(* IEC 61131-3 sources: POMIRTS_lab3/AS/Library/AsHttp, 3 files *)

(* ---- AsHttp.typ ---- *)
(********************************************************************
 * COPYRIGHT -- Bernecker + Rainer
 ********************************************************************
 * Library: AsHttp
 * File: AsHttp.typ
 * Author: B+R
 ********************************************************************
 * Data types of library AsHttp
 ********************************************************************)

TYPE
	httpResponseHeader_t : 	STRUCT  (*response header structure*)
		protocol : STRING[20]; (*HTTP/1.0 or HTTP/1.1*)
		status : STRING[280]; (*HTTP status line e.g. "200 OK" , "404 Not Found"*)
		contentType : STRING[100]; (*MIME type specifying message body, e.g. "text/html"*)
		contentLength : UDINT; (*length of message data, should be equal to responseDataLen, optional input*)
		connection : STRING[80]; (*valid tokens are "Close" or "Keep-Alive", default is "Close"*)
		keepAlive : STRING[80]; (*e.g. "timeout=5, max=100", optional*)
		userLine : ARRAY[0..7]OF httpHeaderLine_t; (*userspecific headerlines, optional*)
		rawHeader : httpRawHeader_t; (*interface to add / get formatted headers, optional*)
	END_STRUCT;
	httpRequestHeader_t : 	STRUCT  (*request header structure*)
		protocol : STRING[20]; (*protocol version e.g. "HTTP/1.0" or "HTTP/1.1", optional input*)
		host : STRING[280]; (*host name or ip address of the server and port number if <> 80, optional input*)
		contentType : STRING[100]; (*MIME type specifying message body, e.g. "text/html", optional input*)
		contentLength : UDINT; (*length of message data, should be equal to requestDataLen, optional input*)
		connection : STRING[80]; (*valid tokens are "Close" or "Keep-Alive", default is "Close", optional input*)
		keepAlive : STRING[80]; (*e.g. "timeout=5, max=100", optional input*)
		userLine : ARRAY[0..7]OF httpHeaderLine_t; (*userspecific headerlines, optional*)
		rawHeader : httpRawHeader_t; (*interface to add / get formatted headers, optional*)
	END_STRUCT;
	httpHeaderLine_t : 	STRUCT  (*structure containing information of one header line*)
		name : STRING[50]; (*header field name, e.g. "User-Agent" to get / set the user-agent header entry*)
		value : STRING[80]; (*header field value, e.g. "B&R Client"*)
	END_STRUCT;
	httpRawHeader_t : 	STRUCT  (*buffer handling structure for raw (formatted) headers*)
		pData : UDINT; (*pointer to data buffer, where the header is copied*)
		dataSize : UDINT; (*max. length of data buffer in bytes*)
		dataLen : UDINT; (*length of the header bytes copied out*)
	END_STRUCT;
	httpStatistics_t : 	STRUCT  (*informational structure*)
		requestCounter : UDINT; (*counts requests*)
		timeOfLastRequest : DATE_AND_TIME; (*timestamp of last request*)
		responseCounter : UDINT; (*counts responses*)
		timeOfLastResponse : DATE_AND_TIME; (*timestamp of last response*)
		errorCounter : UDINT; (*counts errors, e.g. connection errors, aborts *)
		lastError : UDINT; (*error number, if any*)
	END_STRUCT;
END_TYPE

(* ---- AsHttp.fun ---- *)
(********************************************************************
 * COPYRIGHT -- Bernecker + Rainer
 ********************************************************************
 * Library: AsHttp
 * File: AsHttp.fun
 * Author: B+R
 ********************************************************************
 * Functions and function blocks of library AsHttp
 ********************************************************************)

FUNCTION_BLOCK httpService (*offers a webservice ; asynchronous execution*)
	VAR_INPUT
		enable : BOOL; (*enables execution, registers webservice; asynchronous execution*)
		send : BOOL; (*on positive edge response will be sent*)
		abort : BOOL; (*request handling aborts on positive edge*)
		option : UDINT; (*options such as service type, protocol version (HTTP/1.0 , HTTP/1.1), see httpOPTIONS_XXX*)
		pServiceName : UDINT; (*ressource name of webservice, see httpOPTION_SERVICE_TYPE_XXX*)
		pUri : UDINT; (*URI buffer string given as a pointer, an URI may look like "hello.cgi?name=myName"*)
		uriSize : UDINT; (*size of uri data puffer*)
		pRequestHeader : UDINT; (*pointer to httpRequestHeader_t, optional*)
		pRequestData : UDINT; (*request data puffer string given as a pointer*)
		requestDataSize : UDINT; (*size of request data buffer*)
		pResponseHeader : UDINT; (*pointer to httpResponseHeader_t, optional*)
		pResponseData : UDINT; (*response data string given as a pointer*)
		responseDataLen : UDINT; (*length of response data*)
		pStatistics : UDINT; (*pointer to httpStatistics_t, optional*)
		pStruct : UDINT; (*reserve*)
	END_VAR
	VAR_OUTPUT
		status : UINT; (*execution status: ERR_OK, ERR_FUB_ENABLE_FALSE, ERR_FUB_BUSY,0xXXXX = see help*)
		method : UINT; (*method of incoming request, see httpMETHOD_XXX*)
		requestDataLen : UDINT; (*length of request data*)
		phase : UINT; (*current phase of request response handling of the webservice, see httpPHASE_XXX*)
	END_VAR
	VAR
		_i_state : UDINT; (*internal variable*)
		_i_result : UINT; (*internal variable*)
		_ident : UDINT; (*internal variable*)
		_oldEnable : UDINT; (*internal variable*)
		_oldAbort : UDINT; (*internal variable*)
		_oldSend : UDINT; (*internal variable*)
		_state : UDINT; (*internal variable*)
		_internal : UDINT; (*internal variable*)
	END_VAR
END_FUNCTION_BLOCK

FUNCTION_BLOCK httpClient (*sends and recieves HTTP messages (web requests); asynchronous execution*)
	VAR_INPUT
		enable : BOOL; (*enables execution; asynchronous execution*)
		send : BOOL; (*sends request data on positive edge*)
		abort : BOOL; (*disconnects and resets client state on positive edge*)
		option : UDINT; (*options, e.g protocol version (HTTP1.0 / 1.1)*)
		pHost : UDINT; (*host name or ip of server to connect to given as a pointer*)
		hostPort : UINT; (*port number of server to connect to*)
		method : UDINT; (*request method see httpMETHOD_XXX*)
		pUri : UDINT; (*request uri given as a pointer, e.g. "/index.html" or "/hello.cgi?name=myName"*)
		pRequestHeader : UDINT; (*pointer to httpRequestHeader_t, optional*)
		pRequestData : UDINT; (*pointer to request data, typically string data*)
		requestDataLen : UDINT; (*length of request data*)
		pResponseHeader : UDINT; (*pointer to httpResponseHeader_t, optional*)
		pResponseData : UDINT; (*pointer to response data buffer, typically string data*)
		responseDataSize : UDINT; (*size of response data buffer*)
		pStatistics : UDINT; (*pointer to httpStatistics_t, optional*)
		pStruct : UDINT; (*reserve*)
	END_VAR
	VAR_OUTPUT
		status : UINT; (*execution status: ERR_OK, ERR_FUB_ENABLE_FALSE, ERR_FUB_BUSY,
0xXXXX = see help*)
		tcpStatus : UINT; (*status of the tcp connection*)
		httpStatus : UINT; (*status code of response, e.g. 200 for "OK", 404 for "Not Found"*)
		responseDataLen : UDINT; (*length of response (bytes)*)
		phase : UINT; (*current phase of request response handling of the webservice, see httpPHASE_XXX*)
	END_VAR
	VAR
		_i_state : UDINT; (*internal variable*)
		_i_result : UINT; (*internal variable*)
		_ident : UDINT; (*internal variable*)
		_oldEnable : UDINT; (*internal variable*)
		_oldAbort : UDINT; (*internal variable*)
		_oldSend : UDINT; (*internal variable*)
		_state : UDINT; (*internal variable*)
		_internal : UDINT; (*internal variable*)
	END_VAR
END_FUNCTION_BLOCK

FUNCTION_BLOCK httpUtf8ToString (*converts a UTF8 string in string with respect to given code page mapping*)
	VAR_INPUT
		enable : BOOL; (*enables execution*)
		pSrc : UDINT; (*input string (UTF8 encoded), given as a pointer*)
		pDest : UDINT; (*destination buffer*)
		destSize : UDINT; (*size of destination buffer*)
		pMappingTable : UDINT; (*pointer to WSTRING[255],  mapping table for code page, see help*)
	END_VAR
	VAR_OUTPUT
		status : UINT; (*execution status: ERR_OK, ERR_FUB_ENABLE_FALSE, 0xXXXX = see help*)
		destLen : UDINT; (*string length of the string*)
	END_VAR
END_FUNCTION_BLOCK

FUNCTION_BLOCK httpStringToUtf8 (*converts a string in UTF8 string with respect to given code page mapping*)
	VAR_INPUT
		enable : BOOL; (*enables execution*)
		pSrc : UDINT; (*input string, given as a pointer*)
		pDest : UDINT; (*destination buffer*)
		destSize : UDINT; (*size of destination buffer*)
		pMappingTable : UDINT; (*pointer to WSTRING[255],  mapping table for code page, see help*)
	END_VAR
	VAR_OUTPUT
		status : UINT; (*execution status: ERR_OK, ERR_FUB_ENABLE_FALSE, 0xXXXX = see help*)
		destLen : UDINT; (*string length of the UTF8 string*)
	END_VAR
END_FUNCTION_BLOCK

FUNCTION_BLOCK httpUtf8ToWString (*converts a UTF8 encoded string in wide character string*)
	VAR_INPUT
		enable : BOOL; (*enables execution*)
		pSrc : UDINT; (*input string, given as a pointer*)
		pDest : UDINT; (*destination buffer*)
		destSize : UDINT; (*size of destination buffer*)
	END_VAR
	VAR_OUTPUT
		status : UINT; (*execution status: ERR_OK, ERR_FUB_ENABLE_FALSE, 0xXXXX = see help*)
		destLen : UDINT; (*wide character string length*)
	END_VAR
END_FUNCTION_BLOCK

FUNCTION_BLOCK httpWStringToUtf8 (*converts a wide character string in UTF8 string*)
	VAR_INPUT
		enable : BOOL; (*enables execution*)
		pSrc : UDINT; (*input string, given as a pointer*)
		pDest : UDINT; (*destination buffer*)
		destSize : UDINT; (*size of destination buffer*)
	END_VAR
	VAR_OUTPUT
		status : UINT; (*execution status: ERR_OK, ERR_FUB_ENABLE_FALSE, 0xXXXX = see help*)
		destLen : UDINT; (*string length of the UTF8 encoded string*)
	END_VAR
END_FUNCTION_BLOCK

FUNCTION_BLOCK httpDecodeBase64 (*decodes base64 encoded string in binary data or string*)
	VAR_INPUT
		enable : BOOL; (*enables execution*)
		pSrc : UDINT; (*encoded string, given as a pointer*)
		srcLen : UDINT; (*length of encoded string*)
		pDest : UDINT; (*destination buffer, given as a pointer*)
		destSize : UDINT; (*size of destination buffer*)
	END_VAR
	VAR_OUTPUT
		status : UINT; (*execution status: ERR_OK, ERR_FUB_ENABLE_FALSE, 0xXXXX = see help*)
		destLen : UDINT; (*length of decoded data*)
	END_VAR
END_FUNCTION_BLOCK

FUNCTION_BLOCK httpEncodeBase64 (*encodes binary data or a string in a base64 encoded string*)
	VAR_INPUT
		enable : BOOL; (*enables execution*)
		pSrc : UDINT; (*input data, given as a pointer*)
		srcLen : UDINT; (*length of input data*)
		pDest : UDINT; (*destination buffer, given as a pointer*)
		destSize : UDINT; (*size of destination buffer*)
	END_VAR
	VAR_OUTPUT
		status : UINT; (*execution status: ERR_OK, ERR_FUB_ENABLE_FALSE, 0xXXXX = see help*)
		destLen : UDINT; (*length of encoded string*)
	END_VAR
END_FUNCTION_BLOCK

FUNCTION_BLOCK httpEncodeUrl (*encodes special chars in the given string according the URL encoding*)
	VAR_INPUT
		enable : BOOL; (*enables execution*)
		pSrc : UDINT; (*input string, given as a pointer*)
		pDest : UDINT; (*destination buffer, given as a pointer*)
		destSize : UDINT; (*size of destination buffer*)
	END_VAR
	VAR_OUTPUT
		status : UINT; (*execution status: ERR_OK, ERR_FUB_ENABLE_FALSE, 0xXXXX = see help*)
		destLen : UDINT; (*length of encoded string*)
	END_VAR
END_FUNCTION_BLOCK

FUNCTION_BLOCK httpDecodeUrl (*decodes an URL encoded string*)
	VAR_INPUT
		enable : BOOL; (*enables execution*)
		pSrc : UDINT; (*input string, given as a pointer*)
		pDest : UDINT; (*destination buffer, given as a pointer*)
		destSize : UDINT; (*size of destination buffer*)
	END_VAR
	VAR_OUTPUT
		status : UINT; (*execution status: ERR_OK, ERR_FUB_ENABLE_FALSE, 0xXXXX = see help*)
		destLen : UDINT; (*length of decoded string*)
	END_VAR
END_FUNCTION_BLOCK

FUNCTION_BLOCK httpGetParamUrl (*retrieves the string value of the given parameter.*)
	VAR_INPUT
		enable : BOOL; (*enables execution*)
		pSrc : UDINT; (*input string, given as a pointer*)
		pParam : UDINT; (*search string given as a pointer*)
		pValue : UDINT; (*value string buffer given as a pointer*)
		valueSize : UDINT; (*size of value buffer*)
	END_VAR
	VAR_OUTPUT
		status : UINT; (*execution status: ERR_OK, ERR_FUB_ENABLE_FALSE, 0xXXXX = see help*)
		valueLen : UDINT; (*length of value string*)
	END_VAR
END_FUNCTION_BLOCK

FUNCTION_BLOCK httpSetParamUrl (*adds a parameter and its value with respect to URL encoding*)
	VAR_INPUT
		enable : BOOL; (*enables execution*)
		pParam : UDINT; (*name string given as a pointer*)
		pValue : UDINT; (*value string buffer given as a pointer*)
		pDest : UDINT; (*resulting string buffer given as pointer*)
		destSize : UDINT; (*size of destination buffer*)
	END_VAR
	VAR_OUTPUT
		status : UINT; (*execution status: ERR_OK, ERR_FUB_ENABLE_FALSE, 0xXXXX = see help*)
		destLen : UDINT; (*length of resulted string*)
	END_VAR
END_FUNCTION_BLOCK

FUNCTION_BLOCK httpSetBoundary (*adds the boundary information to the HTTP message header*)
	VAR_INPUT
		enable : BOOL; (*enables execution*)
		pStruct : UDINT; (*pointer to the header structure (httpRequestHeader_t or httpResponseHeader_t)*)
		pBoundary : UDINT; (*boundary string given as a pointer. A boundary has no more than 70 chars and is unambiguous*)
	END_VAR
	VAR_OUTPUT
		status : UINT; (*execution status: ERR_OK, ERR_FUB_ENABLE_FALSE, 0xXXXX = see help*)
	END_VAR
END_FUNCTION_BLOCK

FUNCTION_BLOCK httpGetBoundary (*retrieves the boundary value of the given header structure*)
	VAR_INPUT
		enable : BOOL; (*enables execution*)
		pStruct : UDINT; (*pointer to the header structure (httpRequestHeader_t or httpResponseHeader_t)*)
		pBoundary : UDINT; (*boundary string buffer given as a pointer*)
		boundarySize : UDINT; (*size of boundary buffer, preferrably slighly more than 70 bytes*)
	END_VAR
	VAR_OUTPUT
		status : UINT; (*execution status: ERR_OK, ERR_FUB_ENABLE_FALSE, 0xXXXX = see help*)
		boundaryLen : UDINT; (*length of the retrieved boundary if any*)
	END_VAR
END_FUNCTION_BLOCK

FUNCTION_BLOCK httpSetMultipartMessage (*sets respectivly appends a multipart message*)
	VAR_INPUT
		enable : BOOL; (*enables execution*)
		pDest : UDINT; (*destination buffer string given as a pointer*)
		destSize : UDINT; (*size of destination buffer*)
		pBoundary : UDINT; (*boundary string to seperate multipart message given as a pointer*)
		pMessageHeader : UDINT; (*header string given as a pointer, contains header for multipart message, if any*)
		pMessageData : UDINT; (*message body given as a pointer, contains data for multipart message*)
		messageDataLen : UDINT; (*length of message data*)
	END_VAR
	VAR_OUTPUT
		status : UINT; (*execution status: ERR_OK, ERR_FUB_ENABLE_FALSE, 0xXXXX = see help*)
	END_VAR
	VAR
		_messageLen : UDINT; (*internal variable*)
	END_VAR
END_FUNCTION_BLOCK

FUNCTION_BLOCK httpGetMultipartMessage (*gets next multipart message information on each call*)
	VAR_INPUT
		enable : BOOL; (*enables execution*)
		pSrc : UDINT; (*source string given as a pointer, contains one or more multipart messages*)
		pBoundary : UDINT; (*boundary string given as a pointer, seperator of the multipart messages*)
		pMessageHeader : UDINT; (*string buffer for a optional message header given as a pointer*)
		messageHeaderSize : UDINT; (*size of message header buffer*)
		pMessageData : UDINT; (*string buffer for message data given as a pointer*)
		messageDataSize : UDINT; (*size of message data buffer*)
	END_VAR
	VAR_OUTPUT
		status : UINT; (*execution status: ERR_OK, ERR_FUB_ENABLE_FALSE, 0xXXXX = see help*)
		messageHeaderLen : UDINT; (*length of current header, if any*)
		messageDataLen : UDINT; (*length of current data*)
		messageLen : UDINT; (*offset to current message ending*)
	END_VAR
	VAR
		_internal : UDINT; (*internal variable*)
	END_VAR
END_FUNCTION_BLOCK

(* ---- AsHttp.var ---- *)
(********************************************************************
 * COPYRIGHT -- Bernecker + Rainer
 ********************************************************************
 * Library: AsHttp
 * File: AsHttp.var
 * Author: B+R
 ********************************************************************
 * Local variables of library AsHttp
 ********************************************************************)
VAR CONSTANT
	httpERR_BUFFER_SIZE : UINT := 35550; (*buffer is too small*)
	httpERR_DATA_SIZE : UINT := 35551; (*data buffer is too small*)
	httpERR_HEADER_SIZE_RAW : UINT := 35552; (*raw header size buffer is too small or raw header is too long*)
	httpERR_HEADER_SIZE_USERLINE : UINT := 35553; (*any of requested user line is too long for the structure*)
	httpERR_INVALID_PARAM : UINT := 35554; (*check parameters. At least one of needed ones is zero*)
	httpERR_NO_DATA : UINT := 35555; (*no data retrieved*)
	httpERR_METHOD_UNSUPPORTED : UINT := 35556; (*method not supported, supported methods are PUT, POST, GET, DELETE*)
	httpERR_SERVICE_NO_WEBSERVER : UINT := 35557; (*webserver is disabled or not installed, webservice will not be available*)
	httpERR_SERVICE_LINK_FAILED : UINT := 35558; (*webservice could not be registered, check registration*)
	httpERR_CLIENT_ERR_SOCKET_CREATE : UINT := 35559; (*could not create a new socket. Try again later*)
	httpERR_CLIENT_NO_MORE_IDENTS : UINT := 35560; (*too many httpClients enabled, disable unused instances*)
	httpERR_CLIENT_TCP_CONN_CLOSED : UINT := 35561; (*informational, no error: Connection closed. Possible reasons: HTTP/1.0, use of "Connection: close" header, Keep-Alive timeout*)
	httpERR_CLIENT_TCP_CONN_FAILED : UINT := 35562; (*could not connect to given server. Check network parameters and server aviability*)
	httpERR_CLIENT_TCP_INVALID_HOST : UINT := 35563; (*could not resolve name or IP-address of server, check pHost*)
	httpERR_CLIENT_TCP_DISCONNECTED : UINT := 35564; (*lost connection unexpectedly*)
	httpERR_NOT_FOUND : UINT := 35565; (*source string didn't contain parameter*)
	httpERR_ILLEGAL_CHARACTERS : UINT := 35566; (*source contains characters, that couldn't be transformd*)
	httpERR_SYSTEM : UINT := 35579; (*general error, see help*)
	httpMETHOD_GET : UINT := 1; (*request method GET, additional request parameters are part of the URL*)
	httpMETHOD_POST : UINT := 2; (*request method POST, request contains a message body*)
	httpMETHOD_PUT : UINT := 3; (*request method PUT, request contains a message body*)
	httpMETHOD_DELETE : UINT := 4; (*request method DELETE, additional request parameters are part of the URL*)
	httpOPTION_HTTP_10 : UINT := 0; (*use HTTP/1.0 as protocol type*)
	httpOPTION_HTTP_11 : UINT := 1; (*use HTTP/1.1 as protocol type*)
	httpOPTION_SERVICE_TYPE_ROOT : UINT := 4; (*Type of service: root path, e.g. "/basePath", handles requests inside this virtual folder*)
	httpOPTION_SERVICE_TYPE_NAME : UINT := 2; (*Type of service: name, e.g. "hello.cgi", handles requests ending with this name*)
	httpOPTION_SERVICE_TYPE_EXT : UINT := 6; (*Type of service: file extension, e.g. "*.abc" handles requests with file extension ".abc"*)
	httpOPTION_SERVICE_TYPE_LEAF : UINT := 8; (*Type of service: relative path, e.g. "cgi-bin" handles requests in virtual subfolders called "cgi-bin"*)
	httpPHASE_NOT_CONNECTED : UINT := 0; (*not connected*)
	httpPHASE_SENDING : UINT := 1; (*sending a HTTP message*)
	httpPHASE_RECEIVING : UINT := 2; (*receiving a HTTP message*)
	httpPHASE_RECEIVED : UINT := 3; (*HTTP message received *)
	httpPHASE_WAITING : UINT := 4; (*idle state*)
END_VAR
